TYPE "udt_ZoneSafetyInterface"
VERSION : 0.1
// Block: udt_ZoneSafetyInterface
   STRUCT
      Door_NormalStop : Bool;
      Door_SafeStop : Bool;
      Door_Opened : Bool;
      Door_EntryEnable : Bool;
   END_STRUCT;

END_TYPE
